// TIA Portal V19 export
TYPE "Prod_Halted"
// stored: Access Published
   STRUCT
      Code : Int;   // Codice stato interruzione vedere tabella "Prod_Halted_Status_CONST"
      Message_N : Int;   // Numero del messaggio (Alarm /Warning) che identifica la causa dell'interruzione
   END_STRUCT;
END_TYPE
